INTERFACE I_NodeVisitor

METHOD VisitNode
VAR_INPUT
	VisitingNode : I_Node;
END_VAR
END_METHOD

END_INTERFACE

(* stored: Version 1.1.0.1, ProductVersion 3.1.4024.12
   Itf I_NodeVisitor: Id {95baee2a-416d-403f-b4f7-7baf2b821c2b}
   Method VisitNode: Id {1c5e8ee8-5e1d-4274-8f78-d97f85c97ba7} *)
